FUNCTION F_LowerValue : REAL
VAR_INPUT
	Value1																: REAL;
	Value2																: REAL;
END_VAR
VAR
END_VAR

// F_LowerValue
// Rev 1.0 - February 25, 2024

F_LowerValue															:= SEL(Value1 < Value2, Value2, Value1);

END_FUNCTION

(* stored: Version 1.1.0.1, ProductVersion 3.1.4024.12
   POU F_LowerValue: Id {9e88cf8b-2020-4575-a920-4afa8023f33d}, SpecialFunc None *)
